(* Logix 5000 project; controller BTS01 vendor 1 type 14 code 217 rev 32.14; software revision 32.04; part 13 of 15 *)
(* tags used below, declared in another part *)
   AirBlow_Timer : TIMER;
   AirblowPB : BOOL;
   C02S01 : REAL[8];   // 5069-IF8
   C02S02 : REAL[8];   // 5069-OF8
   C02S03 : INT;   // 5069-IB16
   C02S04 : INT;   // 5069-OB16
   C02S05 : INT;   // 5069-OB16
   C02S06 : INT;   // 5069-IB16
   CIP_1_ACTIVE_CIRCUIT : DINT;
   CIP_1_RUN_LATCH : BOOL;
   CIP_1_STEP_ADV_MESSAGE : BOOL;
   CIP_RinseStep_PULSE_ENABLE : BOOL;
   CIP_WashStep_PULSE_ENABLE : BOOL;
   HMI_Alarms_Active : BOOL;
   LT1101 : DTE_SCP_W_LIM;   // Tank 1100 Level Transmitter
   LT1201 : DTE_SCP_W_LIM;   // Tank 1200 Level Transmitter
   TIMERS : TIMER[30];
   TK1100_LVL_SCP : DTE_SCP_W_LIM;   // Tank 1100 Level Remote Display
   TK1200_LVL_SCP : DTE_SCP_W_LIM;   // Tank 1200 Level Remote Display
   TransferEnabled : BOOL;
   TransferSelected : DINT;
   TransferStandby : BOOL;
   UnloadEnabled : BOOL;
   UnloadSelected : DINT;
   UnloadStandby : BOOL;
   V1002 : DTE_Air_Valve_v2;   // CIP Bypass Valve
   V1002_CIP_ENABLE : BOOL;
   V1002_CIP_PULSE : BOOL;
   V1002_Desc : STRING;
   V1002_PIDName : STRING;
   V1003 : DTE_Air_Valve_v2;   // Filler Valve
   V1003_CIP_ENABLE : BOOL;
   V1003_CIP_PULSE : BOOL;
   V1003_Desc : STRING;
   V1003_PIDName : STRING;
   V1004 : DTE_Air_Valve_v2;   // Filler Valve
   V1004_CIP_ENABLE : BOOL;
   V1004_CIP_PULSE : BOOL;
   V1004_Desc : STRING;
   V1004_PIDName : STRING;
   V1005 : DTE_Air_Valve_v2;   // Filler Valve
   V1005_CIP_ENABLE : BOOL;
   V1005_CIP_PULSE : BOOL;
   V1005_Desc : STRING;
   V1005_PIDName : STRING;
   V1006 : DTE_Air_Valve_v2;   // Filler Valve
   V1006_CIP_ENABLE : BOOL;
   V1006_CIP_PULSE : BOOL;
   V1006_Desc : STRING;
   V1006_PIDName : STRING;
   V1007 : DTE_Air_Valve_v2;   // Filler Valve
   V1007_CIP_ENABLE : BOOL;
   V1007_CIP_PULSE : BOOL;
   V1007_Desc : STRING;
   V1007_PIDName : STRING;
   V1101 : DTE_Air_Valve_v2;   // Tank 1100 Fill Valve
   V1101_CIP_ENABLE : BOOL;
   V1101_CIP_PULSE : BOOL;
   V1101_Desc : STRING;
   V1101_PIDName : STRING;
   V1102 : DTE_Air_Valve_v2;   // Tank 1100 Discharge Valve
   V1102_CIP_ENABLE : BOOL;
   V1102_CIP_PULSE : BOOL;
   V1102_Desc : STRING;
   V1102_PIDName : STRING;
   V1103 : DTE_Air_Valve_v2;   // Tank 1100 Line Valve
   V1103_CIP_ENABLE : BOOL;
   V1103_CIP_PULSE : BOOL;
   V1103_Desc : STRING;
   V1103_PIDName : STRING;
   V1201 : DTE_Air_Valve_v2;   // Tank 1200 Fill Valve
   V1201_CIP_ENABLE : BOOL;
   V1201_CIP_PULSE : BOOL;
   V1201_Desc : STRING;
   V1201_PIDName : STRING;
   V1202 : DTE_Air_Valve_v2;   // Tank 1200 Discharge Valve
   V1202_CIP_ENABLE : BOOL;
   V1202_CIP_PULSE : BOOL;
   V1202_Desc : STRING;
   V1202_PIDName : STRING;
   V1203 : DTE_Air_Valve_v2;   // Tank 1200 Line Valve
   V1203_CIP_ENABLE : BOOL;
   V1203_CIP_PULSE : BOOL;
   V1203_Desc : STRING;
   V1203_PIDName : STRING;
   VFD1001_SCP : DTE_SCP_W_LIM;   // Bowl Chopper Disc Speed Reference
   VFD1002_SCP : DTE_SCP_W_LIM;   // Dressing Tank Disc Speed Reference
   VFD1003_SCP : DTE_SCP_W_LIM;   // CIP Return Pump Speed Reference
   VFD1004_SCP : DTE_SCP_W_LIM;   // Filler CIP Return Pump Speed Reference
   VFD1101_SCP : DTE_SCP_W_LIM;   // Tank 1100 Agitator Speed Reference
   VFD1201_SCP : DTE_SCP_W_LIM;   // Tank 1200 Agitator Speed Reference
(* MainProgram, continued *)

ROUTINE R01_Digital_Input   (* ladder *)
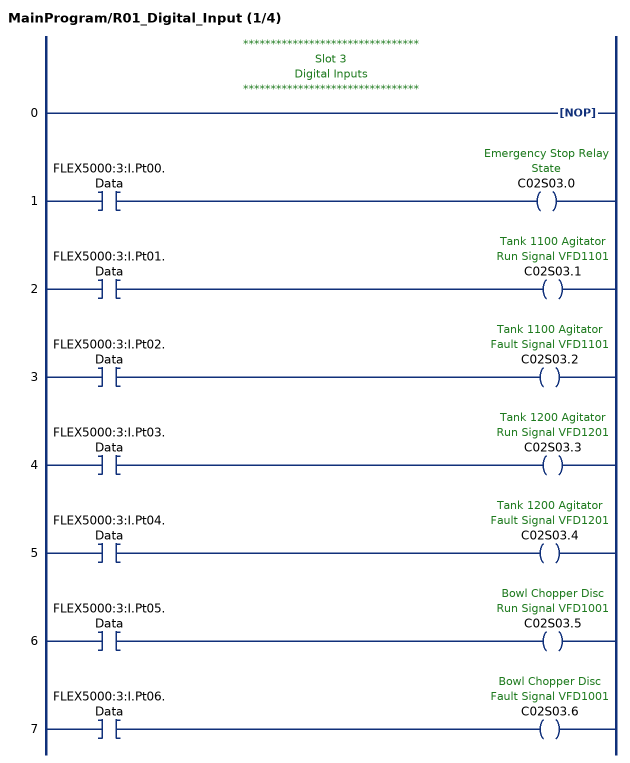
   // ********************************
   // Slot 3
   // Digital Inputs
   // ********************************
   0: NOP();
   1: XIC(FLEX5000:3:I.Pt00.Data)OTE(C02S03.0);
   2: XIC(FLEX5000:3:I.Pt01.Data)OTE(C02S03.1);
   3: XIC(FLEX5000:3:I.Pt02.Data)OTE(C02S03.2);
   4: XIC(FLEX5000:3:I.Pt03.Data)OTE(C02S03.3);
   5: XIC(FLEX5000:3:I.Pt04.Data)OTE(C02S03.4);
   6: XIC(FLEX5000:3:I.Pt05.Data)OTE(C02S03.5);
   7: XIC(FLEX5000:3:I.Pt06.Data)OTE(C02S03.6);
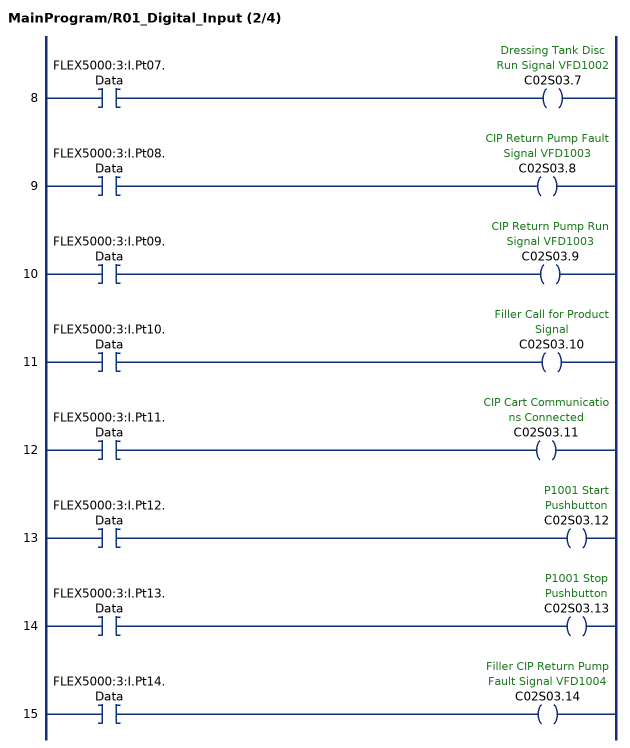
   8: XIC(FLEX5000:3:I.Pt07.Data)OTE(C02S03.7);
   9: XIC(FLEX5000:3:I.Pt08.Data)OTE(C02S03.8);
   10: XIC(FLEX5000:3:I.Pt09.Data)OTE(C02S03.9);
   11: XIC(FLEX5000:3:I.Pt10.Data)OTE(C02S03.10);
   12: XIC(FLEX5000:3:I.Pt11.Data)OTE(C02S03.11);
   13: XIC(FLEX5000:3:I.Pt12.Data)OTE(C02S03.12);
   14: XIC(FLEX5000:3:I.Pt13.Data)OTE(C02S03.13);
   15: XIC(FLEX5000:3:I.Pt14.Data)OTE(C02S03.14);
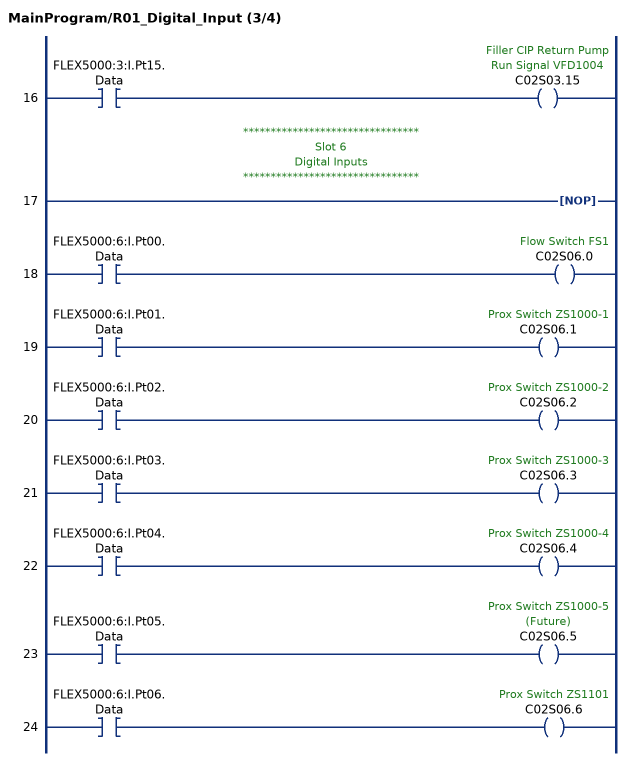
   16: XIC(FLEX5000:3:I.Pt15.Data)OTE(C02S03.15);
   // ********************************
   // Slot 6
   // Digital Inputs
   // ********************************
   17: NOP();
   18: XIC(FLEX5000:6:I.Pt00.Data)OTE(C02S06.0);
   19: XIC(FLEX5000:6:I.Pt01.Data)OTE(C02S06.1);
   20: XIC(FLEX5000:6:I.Pt02.Data)OTE(C02S06.2);
   21: XIC(FLEX5000:6:I.Pt03.Data)OTE(C02S06.3);
   22: XIC(FLEX5000:6:I.Pt04.Data)OTE(C02S06.4);
   23: XIC(FLEX5000:6:I.Pt05.Data)OTE(C02S06.5);
   24: XIC(FLEX5000:6:I.Pt06.Data)OTE(C02S06.6);
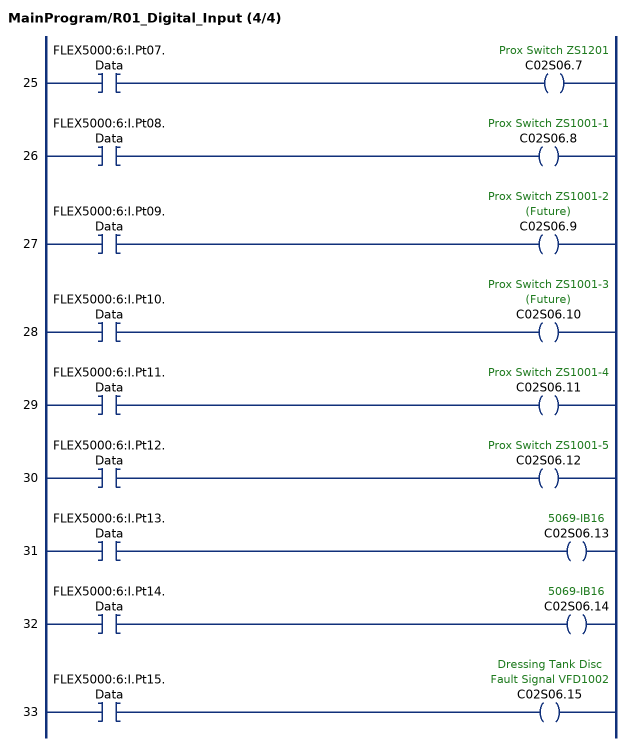
   25: XIC(FLEX5000:6:I.Pt07.Data)OTE(C02S06.7);
   26: XIC(FLEX5000:6:I.Pt08.Data)OTE(C02S06.8);
   27: XIC(FLEX5000:6:I.Pt09.Data)OTE(C02S06.9);
   28: XIC(FLEX5000:6:I.Pt10.Data)OTE(C02S06.10);
   29: XIC(FLEX5000:6:I.Pt11.Data)OTE(C02S06.11);
   30: XIC(FLEX5000:6:I.Pt12.Data)OTE(C02S06.12);
   31: XIC(FLEX5000:6:I.Pt13.Data)OTE(C02S06.13);
   32: XIC(FLEX5000:6:I.Pt14.Data)OTE(C02S06.14);
   33: XIC(FLEX5000:6:I.Pt15.Data)OTE(C02S06.15);
END_ROUTINE

ROUTINE R02_Digital_Output   (* ladder *)
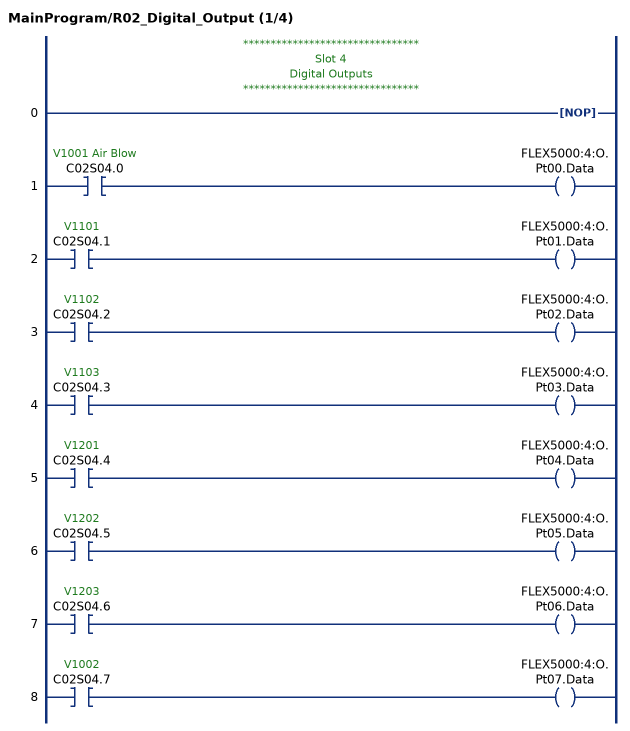
   // ********************************
   // Slot 4
   // Digital Outputs
   // ********************************
   0: NOP();
   1: XIC(C02S04.0)OTE(FLEX5000:4:O.Pt00.Data);
   2: XIC(C02S04.1)OTE(FLEX5000:4:O.Pt01.Data);
   3: XIC(C02S04.2)OTE(FLEX5000:4:O.Pt02.Data);
   4: XIC(C02S04.3)OTE(FLEX5000:4:O.Pt03.Data);
   5: XIC(C02S04.4)OTE(FLEX5000:4:O.Pt04.Data);
   6: XIC(C02S04.5)OTE(FLEX5000:4:O.Pt05.Data);
   7: XIC(C02S04.6)OTE(FLEX5000:4:O.Pt06.Data);
   8: XIC(C02S04.7)OTE(FLEX5000:4:O.Pt07.Data);
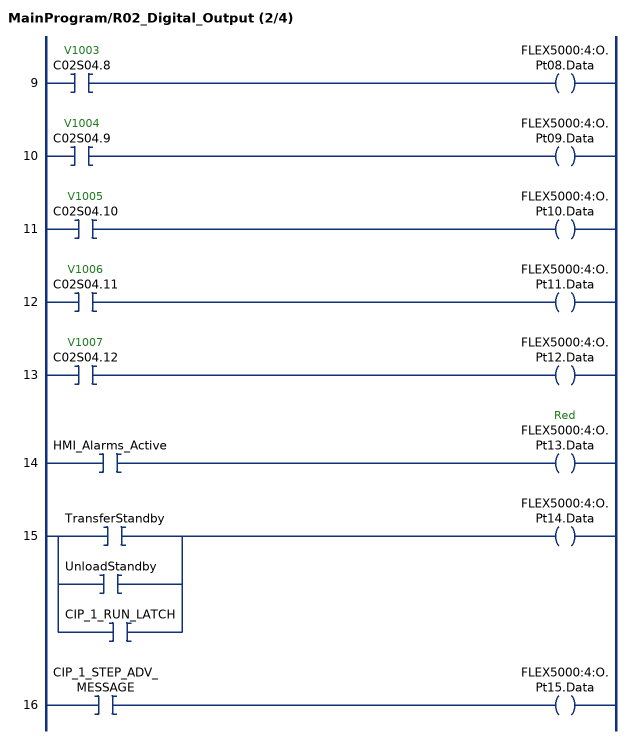
   9: XIC(C02S04.8)OTE(FLEX5000:4:O.Pt08.Data);
   10: XIC(C02S04.9)OTE(FLEX5000:4:O.Pt09.Data);
   11: XIC(C02S04.10)OTE(FLEX5000:4:O.Pt10.Data);
   12: XIC(C02S04.11)OTE(FLEX5000:4:O.Pt11.Data);
   13: XIC(C02S04.12)OTE(FLEX5000:4:O.Pt12.Data);
   14: XIC(HMI_Alarms_Active)OTE(FLEX5000:4:O.Pt13.Data);
   15: [XIC(TransferStandby) ,XIC(UnloadStandby) ,XIC(CIP_1_RUN_LATCH) ]OTE(FLEX5000:4:O.Pt14.Data);
   16: XIC(CIP_1_STEP_ADV_MESSAGE)OTE(FLEX5000:4:O.Pt15.Data);
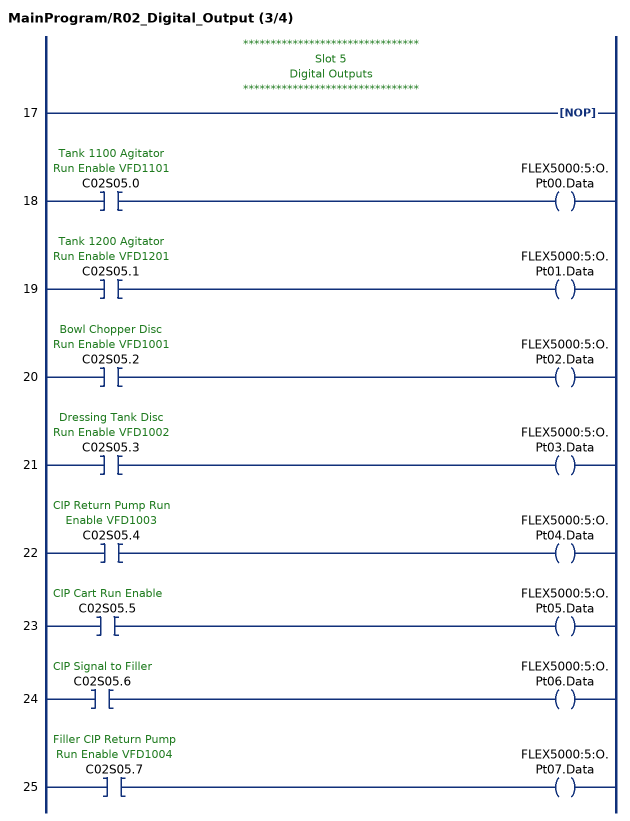
   // ********************************
   // Slot 5
   // Digital Outputs
   // ********************************
   17: NOP();
   18: XIC(C02S05.0)OTE(FLEX5000:5:O.Pt00.Data);
   19: XIC(C02S05.1)OTE(FLEX5000:5:O.Pt01.Data);
   20: XIC(C02S05.2)OTE(FLEX5000:5:O.Pt02.Data);
   21: XIC(C02S05.3)OTE(FLEX5000:5:O.Pt03.Data);
   22: XIC(C02S05.4)OTE(FLEX5000:5:O.Pt04.Data);
   23: XIC(C02S05.5)OTE(FLEX5000:5:O.Pt05.Data);
   24: XIC(C02S05.6)OTE(FLEX5000:5:O.Pt06.Data);
   25: XIC(C02S05.7)OTE(FLEX5000:5:O.Pt07.Data);
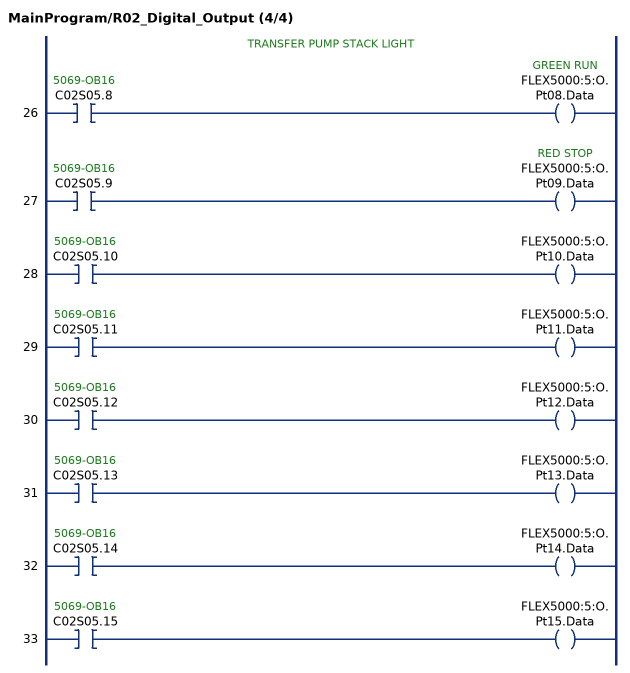
   // TRANSFER PUMP STACK LIGHT
   26: XIC(C02S05.8)OTE(FLEX5000:5:O.Pt08.Data);
   27: XIC(C02S05.9)OTE(FLEX5000:5:O.Pt09.Data);
   28: XIC(C02S05.10)OTE(FLEX5000:5:O.Pt10.Data);
   29: XIC(C02S05.11)OTE(FLEX5000:5:O.Pt11.Data);
   30: XIC(C02S05.12)OTE(FLEX5000:5:O.Pt12.Data);
   31: XIC(C02S05.13)OTE(FLEX5000:5:O.Pt13.Data);
   32: XIC(C02S05.14)OTE(FLEX5000:5:O.Pt14.Data);
   33: XIC(C02S05.15)OTE(FLEX5000:5:O.Pt15.Data);
END_ROUTINE

ROUTINE R03_Analog_Input   (* ladder *)
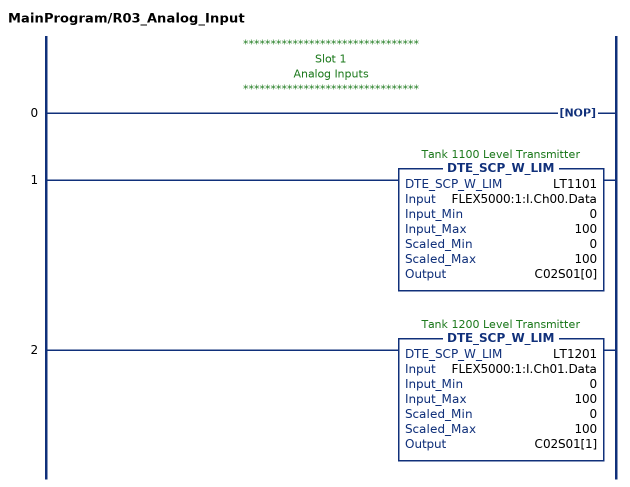
   // ********************************
   // Slot 1
   // Analog Inputs
   // ********************************
   0: NOP();
   1: DTE_SCP_W_LIM(LT1101,FLEX5000:1:I.Ch00.Data,0,100,0,100,C02S01[0]);
   2: DTE_SCP_W_LIM(LT1201,FLEX5000:1:I.Ch01.Data,0,100,0,100,C02S01[1]);
END_ROUTINE

ROUTINE R04_Analog_Output   (* ladder *)
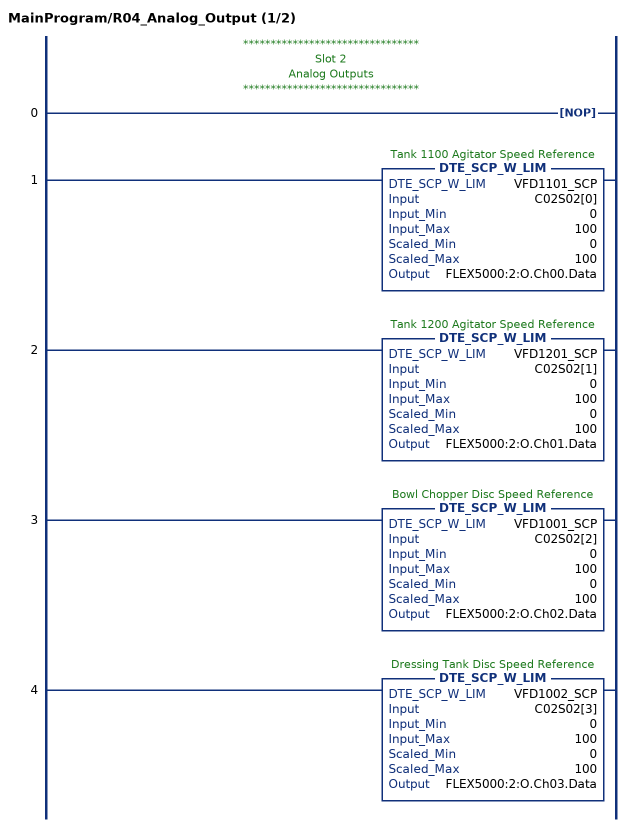
   // ********************************
   // Slot 2
   // Analog Outputs
   // ********************************
   0: NOP();
   1: DTE_SCP_W_LIM(VFD1101_SCP,C02S02[0],0,100,0,100,FLEX5000:2:O.Ch00.Data);
   2: DTE_SCP_W_LIM(VFD1201_SCP,C02S02[1],0,100,0,100,FLEX5000:2:O.Ch01.Data);
   3: DTE_SCP_W_LIM(VFD1001_SCP,C02S02[2],0,100,0,100,FLEX5000:2:O.Ch02.Data);
   4: DTE_SCP_W_LIM(VFD1002_SCP,C02S02[3],0,100,0,100,FLEX5000:2:O.Ch03.Data);
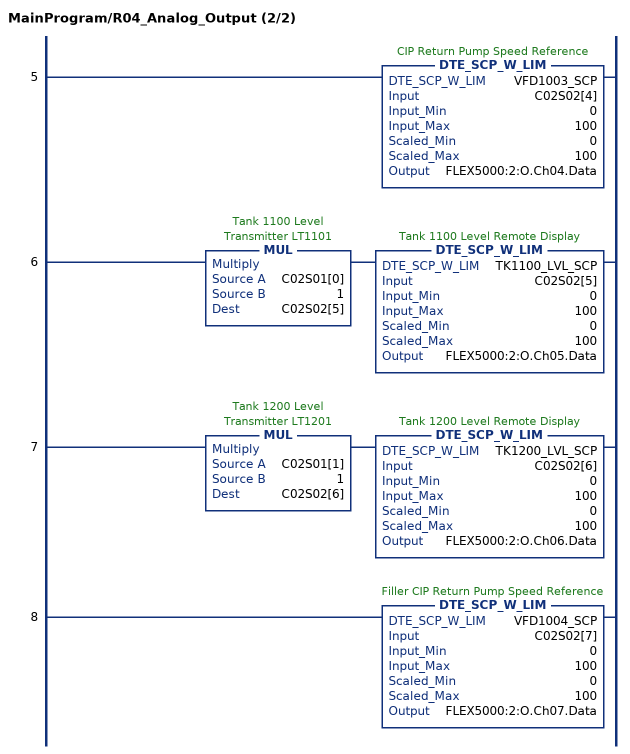
   5: DTE_SCP_W_LIM(VFD1003_SCP,C02S02[4],0,100,0,100,FLEX5000:2:O.Ch04.Data);
   6: MUL(C02S01[0],1,C02S02[5])DTE_SCP_W_LIM(TK1100_LVL_SCP,C02S02[5],0,100,0,100,FLEX5000:2:O.Ch05.Data);
   7: MUL(C02S01[1],1,C02S02[6])DTE_SCP_W_LIM(TK1200_LVL_SCP,C02S02[6],0,100,0,100,FLEX5000:2:O.Ch06.Data);
   8: DTE_SCP_W_LIM(VFD1004_SCP,C02S02[7],0,100,0,100,FLEX5000:2:O.Ch07.Data);
END_ROUTINE

ROUTINE R05_Valves   (* ladder *)
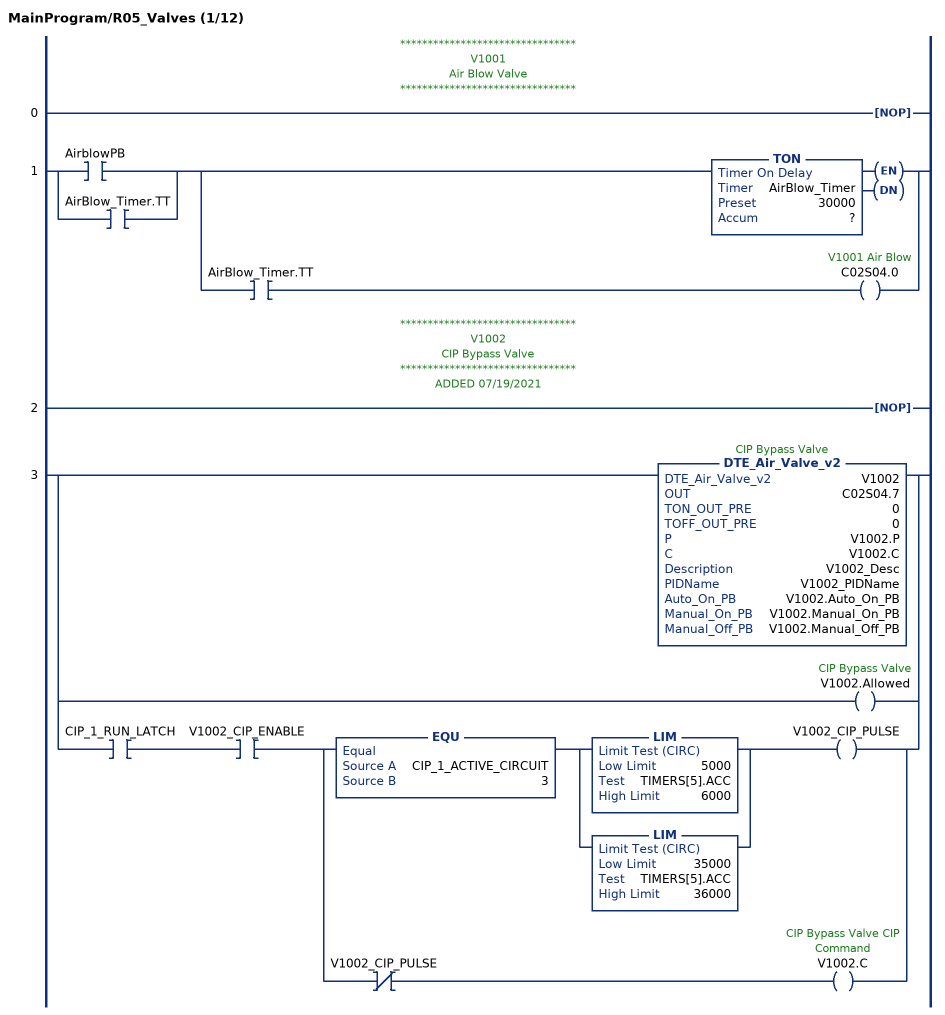
   // ********************************
   // V1001
   // Air Blow Valve
   // ********************************
   0: NOP();
   1: [XIC(AirblowPB) ,XIC(AirBlow_Timer.TT) ][TON(AirBlow_Timer,?,?) ,XIC(AirBlow_Timer.TT) OTE(C02S04.0) ];
   // ********************************
   // V1002
   // CIP Bypass Valve
   // ********************************
   // ADDED 07/19/2021
   2: NOP();
   3: [DTE_Air_Valve_v2(V1002,C02S04.7,0,0,V1002.P,V1002.C,V1002_Desc,V1002_PIDName,V1002.Auto_On_PB,V1002.Manual_On_PB,V1002.Manual_Off_PB) ,OTE(V1002.Allowed) ,XIC(CIP_1_RUN_LATCH) XIC(V1002_CIP_ENABLE) [EQU(CIP_1_ACTIVE_CIRCUIT,3) [LIM(5000,TIMERS[5].ACC,6000) ,LIM(35000,TIMERS[5].ACC,36000) ] OTE(V1002_CIP_PULSE) ,XIO(V1002_CIP_PULSE) OTE(V1002.C) ] ];
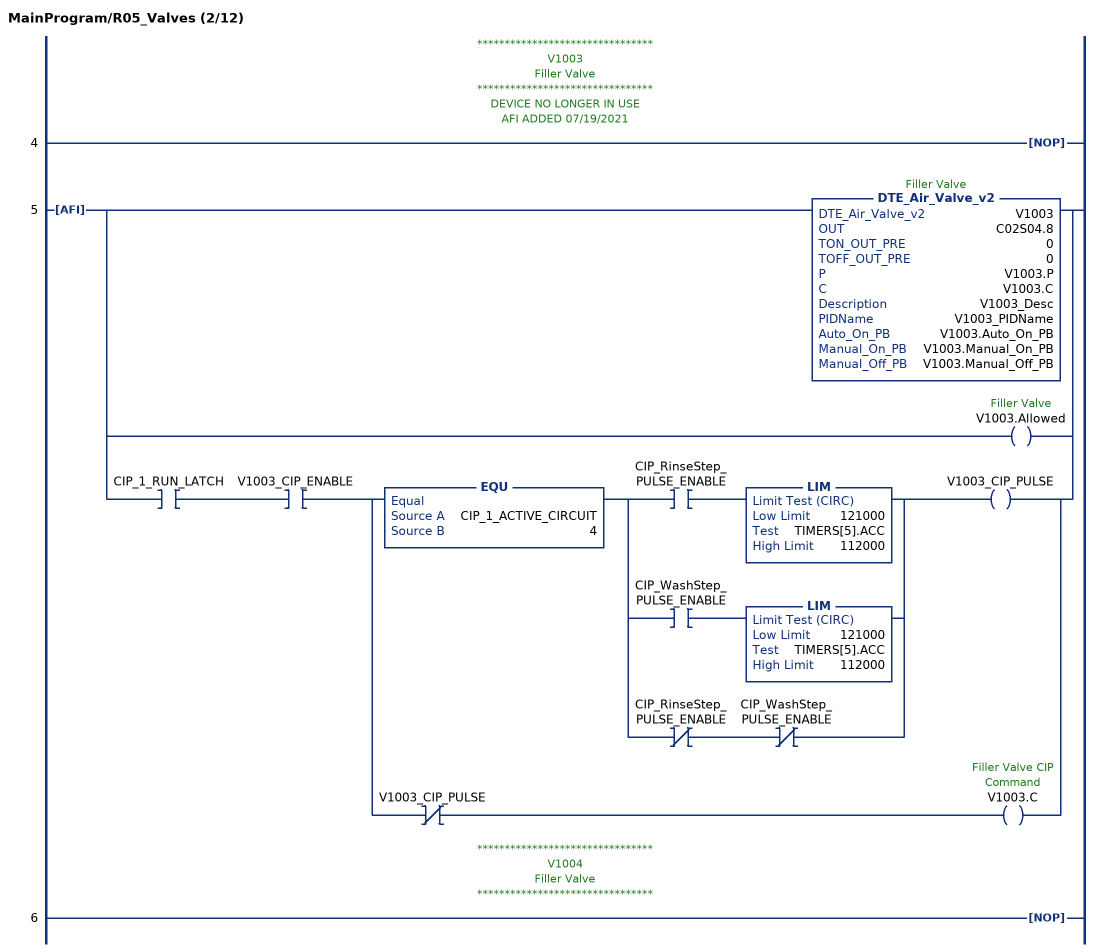
   // ********************************
   // V1003
   // Filler Valve
   // ********************************
   // DEVICE NO LONGER IN USE
   // AFI ADDED 07/19/2021
   4: NOP();
   5: AFI()[DTE_Air_Valve_v2(V1003,C02S04.8,0,0,V1003.P,V1003.C,V1003_Desc,V1003_PIDName,V1003.Auto_On_PB,V1003.Manual_On_PB,V1003.Manual_Off_PB) ,OTE(V1003.Allowed) ,XIC(CIP_1_RUN_LATCH) XIC(V1003_CIP_ENABLE) [EQU(CIP_1_ACTIVE_CIRCUIT,4) [XIC(CIP_RinseStep_PULSE_ENABLE) LIM(121000,TIMERS[5].ACC,112000) ,XIC(CIP_WashStep_PULSE_ENABLE) LIM(121000,TIMERS[5].ACC,112000) ,XIO(CIP_RinseStep_PULSE_ENABLE) XIO(CIP_WashStep_PULSE_ENABLE) ] OTE(V1003_CIP_PULSE) ,XIO(V1003_CIP_PULSE) OTE(V1003.C) ] ];
   // ********************************
   // V1004
   // Filler Valve
   // ********************************
   6: NOP();
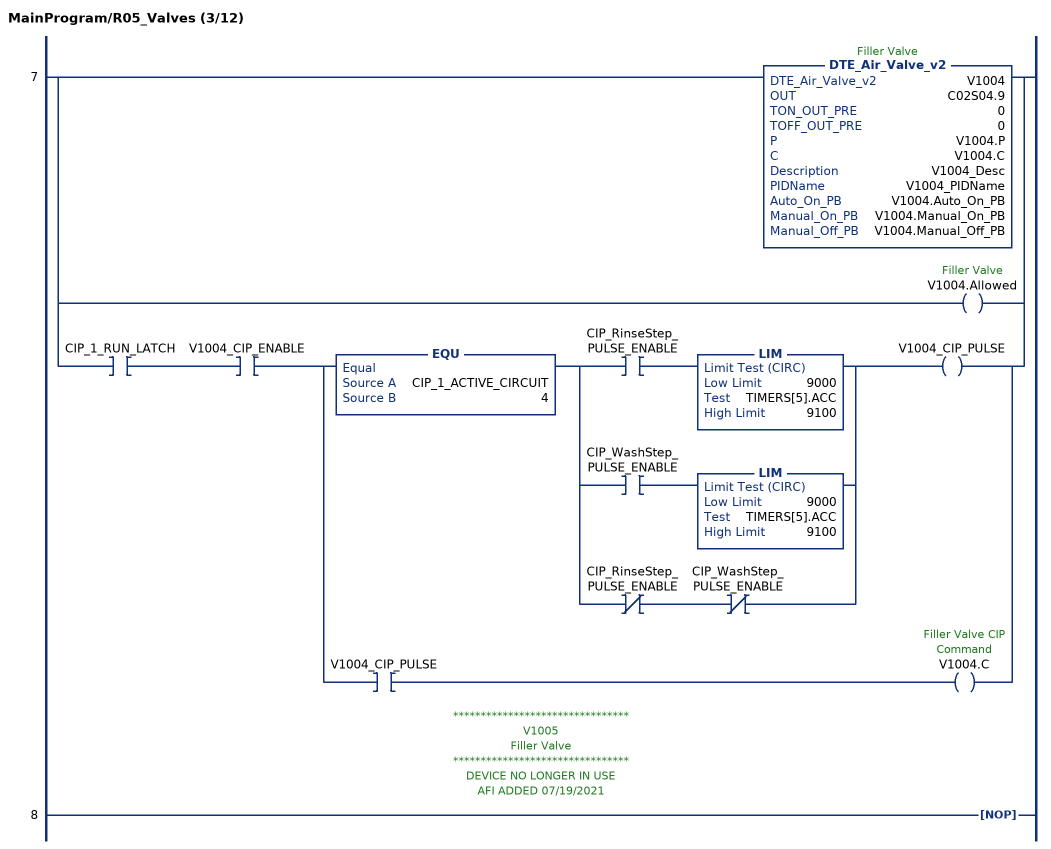
   7: [DTE_Air_Valve_v2(V1004,C02S04.9,0,0,V1004.P,V1004.C,V1004_Desc,V1004_PIDName,V1004.Auto_On_PB,V1004.Manual_On_PB,V1004.Manual_Off_PB) ,OTE(V1004.Allowed) ,XIC(CIP_1_RUN_LATCH) XIC(V1004_CIP_ENABLE) [EQU(CIP_1_ACTIVE_CIRCUIT,4) [XIC(CIP_RinseStep_PULSE_ENABLE) LIM(9000,TIMERS[5].ACC,9100) ,XIC(CIP_WashStep_PULSE_ENABLE) LIM(9000,TIMERS[5].ACC,9100) ,XIO(CIP_RinseStep_PULSE_ENABLE) XIO(CIP_WashStep_PULSE_ENABLE) ] OTE(V1004_CIP_PULSE) ,XIC(V1004_CIP_PULSE) OTE(V1004.C) ] ];
   // ********************************
   // V1005
   // Filler Valve
   // ********************************
   // DEVICE NO LONGER IN USE
   // AFI ADDED 07/19/2021
   8: NOP();
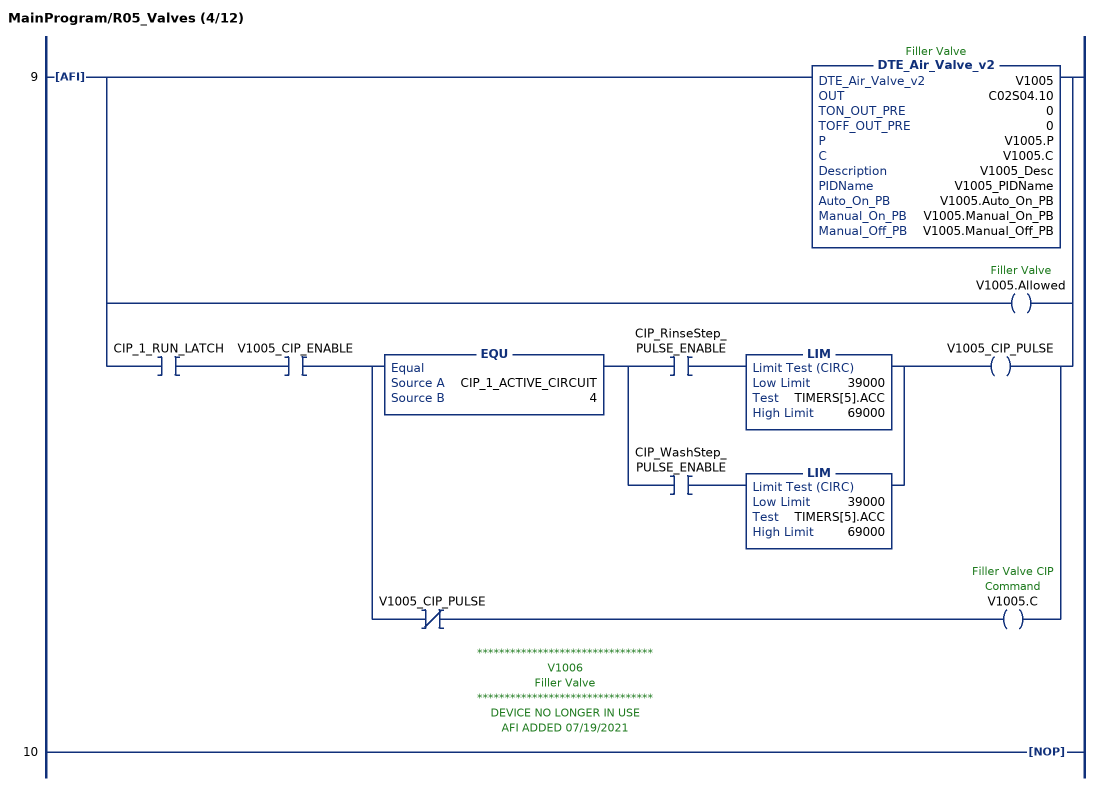
   9: AFI()[DTE_Air_Valve_v2(V1005,C02S04.10,0,0,V1005.P,V1005.C,V1005_Desc,V1005_PIDName,V1005.Auto_On_PB,V1005.Manual_On_PB,V1005.Manual_Off_PB) ,OTE(V1005.Allowed) ,XIC(CIP_1_RUN_LATCH) XIC(V1005_CIP_ENABLE) [EQU(CIP_1_ACTIVE_CIRCUIT,4) [XIC(CIP_RinseStep_PULSE_ENABLE) LIM(39000,TIMERS[5].ACC,69000) ,XIC(CIP_WashStep_PULSE_ENABLE) LIM(39000,TIMERS[5].ACC,69000) ] OTE(V1005_CIP_PULSE) ,XIO(V1005_CIP_PULSE) OTE(V1005.C) ] ];
   // ********************************
   // V1006
   // Filler Valve
   // ********************************
   // DEVICE NO LONGER IN USE
   // AFI ADDED 07/19/2021
   10: NOP();
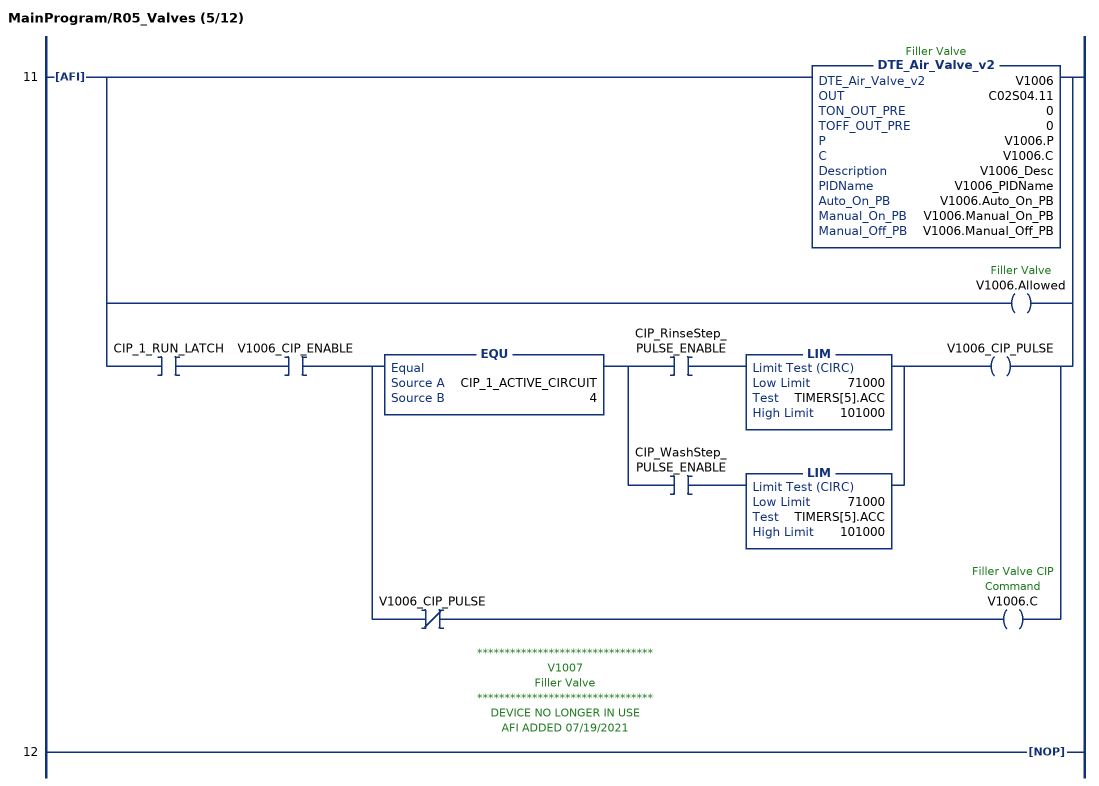
   11: AFI()[DTE_Air_Valve_v2(V1006,C02S04.11,0,0,V1006.P,V1006.C,V1006_Desc,V1006_PIDName,V1006.Auto_On_PB,V1006.Manual_On_PB,V1006.Manual_Off_PB) ,OTE(V1006.Allowed) ,XIC(CIP_1_RUN_LATCH) XIC(V1006_CIP_ENABLE) [EQU(CIP_1_ACTIVE_CIRCUIT,4) [XIC(CIP_RinseStep_PULSE_ENABLE) LIM(71000,TIMERS[5].ACC,101000) ,XIC(CIP_WashStep_PULSE_ENABLE) LIM(71000,TIMERS[5].ACC,101000) ] OTE(V1006_CIP_PULSE) ,XIO(V1006_CIP_PULSE) OTE(V1006.C) ] ];
   // ********************************
   // V1007
   // Filler Valve
   // ********************************
   // DEVICE NO LONGER IN USE
   // AFI ADDED 07/19/2021
   12: NOP();
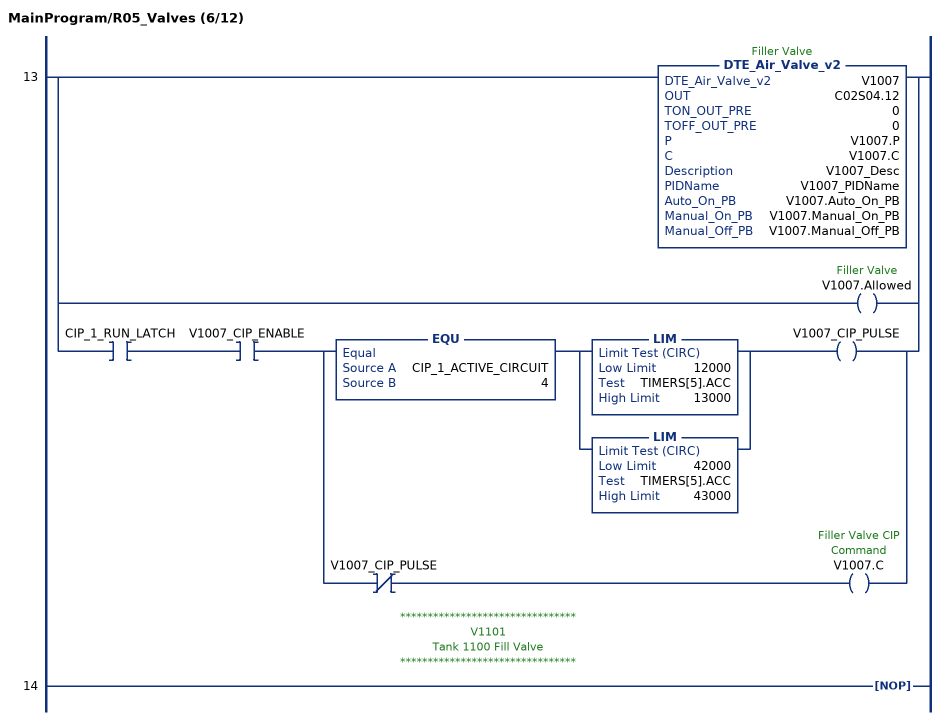
   13: [DTE_Air_Valve_v2(V1007,C02S04.12,0,0,V1007.P,V1007.C,V1007_Desc,V1007_PIDName,V1007.Auto_On_PB,V1007.Manual_On_PB,V1007.Manual_Off_PB) ,OTE(V1007.Allowed) ,XIC(CIP_1_RUN_LATCH) XIC(V1007_CIP_ENABLE) [EQU(CIP_1_ACTIVE_CIRCUIT,4) [LIM(12000,TIMERS[5].ACC,13000) ,LIM(42000,TIMERS[5].ACC,43000) ] OTE(V1007_CIP_PULSE) ,XIO(V1007_CIP_PULSE) OTE(V1007.C) ] ];
   // ********************************
   // V1101
   // Tank 1100 Fill Valve
   // ********************************
   14: NOP();
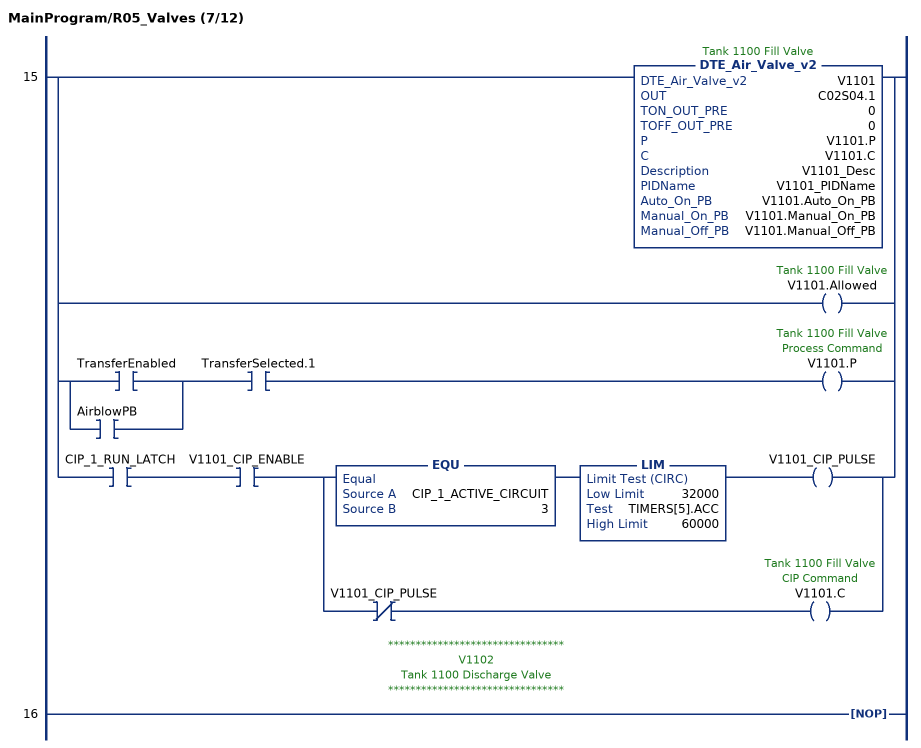
   15: [DTE_Air_Valve_v2(V1101,C02S04.1,0,0,V1101.P,V1101.C,V1101_Desc,V1101_PIDName,V1101.Auto_On_PB,V1101.Manual_On_PB,V1101.Manual_Off_PB) ,OTE(V1101.Allowed) ,[XIC(TransferEnabled) ,XIC(AirblowPB) ] XIC(TransferSelected.1) OTE(V1101.P) ,XIC(CIP_1_RUN_LATCH) XIC(V1101_CIP_ENABLE) [EQU(CIP_1_ACTIVE_CIRCUIT,3) LIM(32000,TIMERS[5].ACC,60000) OTE(V1101_CIP_PULSE) ,XIO(V1101_CIP_PULSE) OTE(V1101.C) ] ];
   // ********************************
   // V1102
   // Tank 1100 Discharge Valve
   // ********************************
   16: NOP();
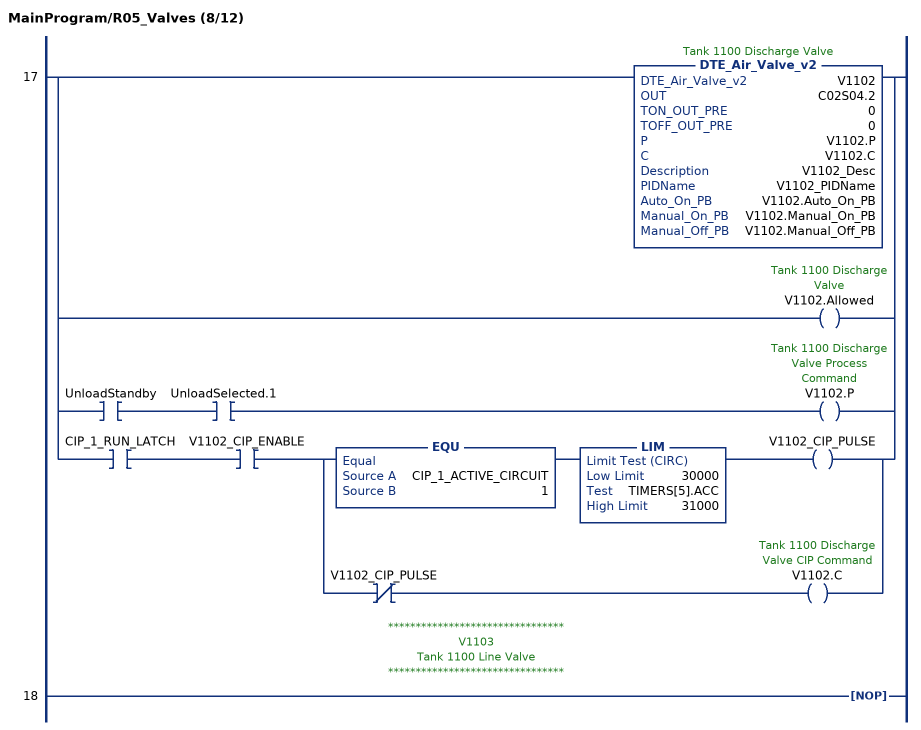
   17: [DTE_Air_Valve_v2(V1102,C02S04.2,0,0,V1102.P,V1102.C,V1102_Desc,V1102_PIDName,V1102.Auto_On_PB,V1102.Manual_On_PB,V1102.Manual_Off_PB) ,OTE(V1102.Allowed) ,XIC(UnloadStandby) XIC(UnloadSelected.1) OTE(V1102.P) ,XIC(CIP_1_RUN_LATCH) XIC(V1102_CIP_ENABLE) [EQU(CIP_1_ACTIVE_CIRCUIT,1) LIM(30000,TIMERS[5].ACC,31000) OTE(V1102_CIP_PULSE) ,XIO(V1102_CIP_PULSE) OTE(V1102.C) ] ];
   // ********************************
   // V1103
   // Tank 1100 Line Valve
   // ********************************
   18: NOP();
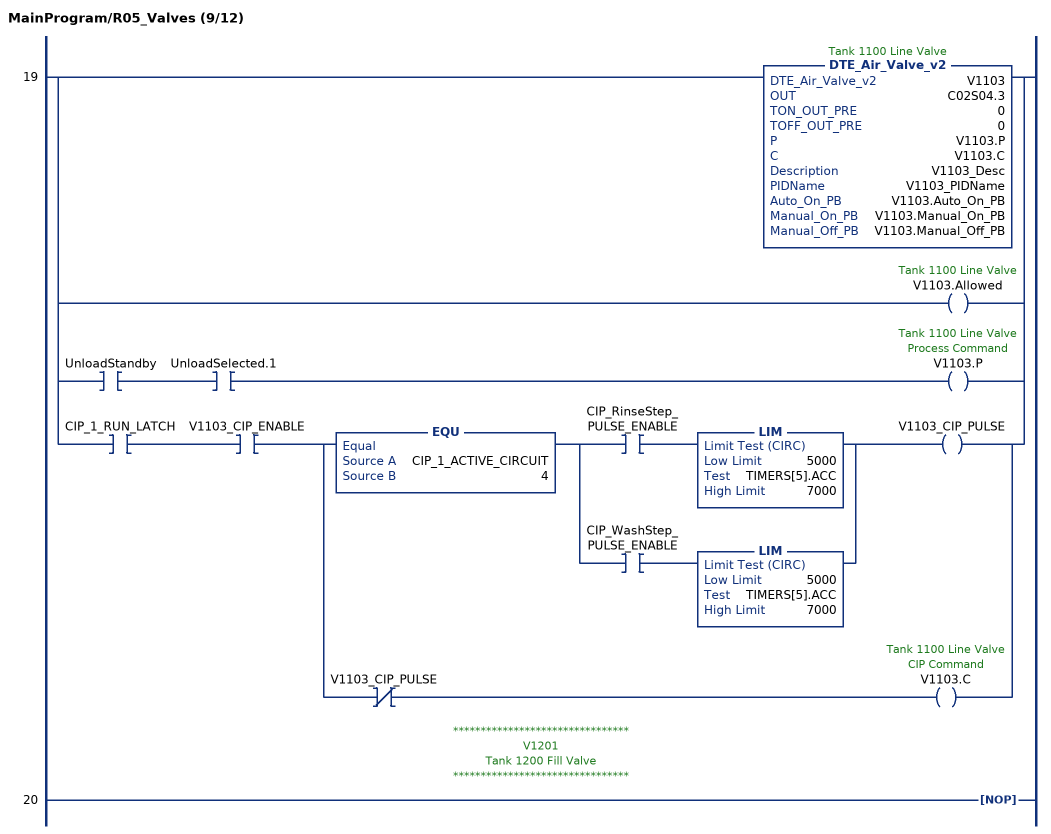
   19: [DTE_Air_Valve_v2(V1103,C02S04.3,0,0,V1103.P,V1103.C,V1103_Desc,V1103_PIDName,V1103.Auto_On_PB,V1103.Manual_On_PB,V1103.Manual_Off_PB) ,OTE(V1103.Allowed) ,XIC(UnloadStandby) XIC(UnloadSelected.1) OTE(V1103.P) ,XIC(CIP_1_RUN_LATCH) XIC(V1103_CIP_ENABLE) [EQU(CIP_1_ACTIVE_CIRCUIT,4) [XIC(CIP_RinseStep_PULSE_ENABLE) LIM(5000,TIMERS[5].ACC,7000) ,XIC(CIP_WashStep_PULSE_ENABLE) LIM(5000,TIMERS[5].ACC,7000) ] OTE(V1103_CIP_PULSE) ,XIO(V1103_CIP_PULSE) OTE(V1103.C) ] ];
   // ********************************
   // V1201
   // Tank 1200 Fill Valve
   // ********************************
   20: NOP();
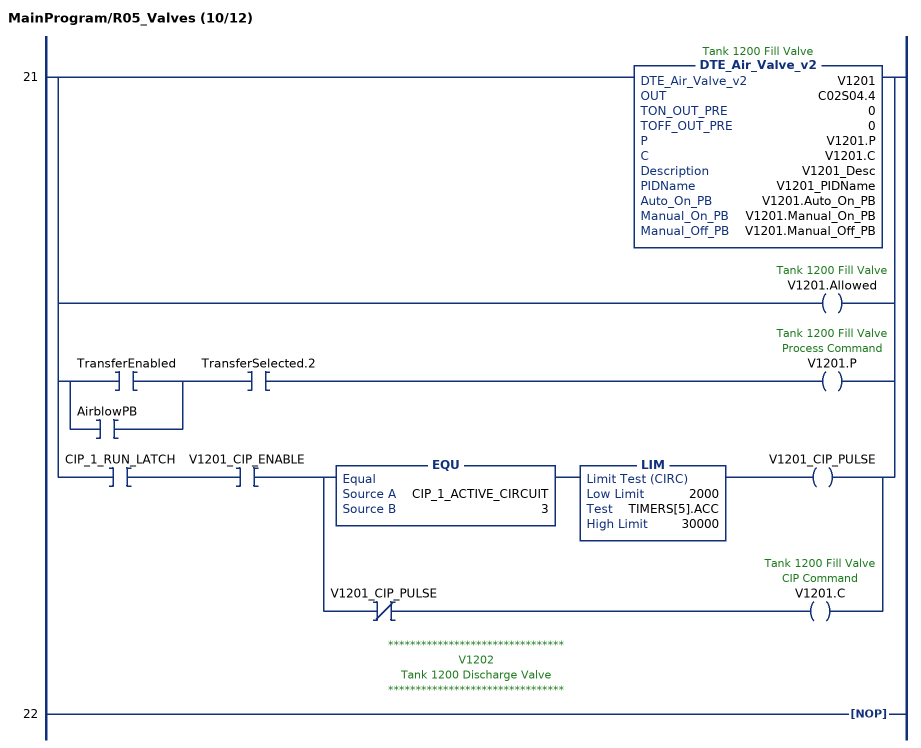
   21: [DTE_Air_Valve_v2(V1201,C02S04.4,0,0,V1201.P,V1201.C,V1201_Desc,V1201_PIDName,V1201.Auto_On_PB,V1201.Manual_On_PB,V1201.Manual_Off_PB) ,OTE(V1201.Allowed) ,[XIC(TransferEnabled) ,XIC(AirblowPB) ] XIC(TransferSelected.2) OTE(V1201.P) ,XIC(CIP_1_RUN_LATCH) XIC(V1201_CIP_ENABLE) [EQU(CIP_1_ACTIVE_CIRCUIT,3) LIM(2000,TIMERS[5].ACC,30000) OTE(V1201_CIP_PULSE) ,XIO(V1201_CIP_PULSE) OTE(V1201.C) ] ];
   // ********************************
   // V1202
   // Tank 1200 Discharge Valve
   // ********************************
   22: NOP();
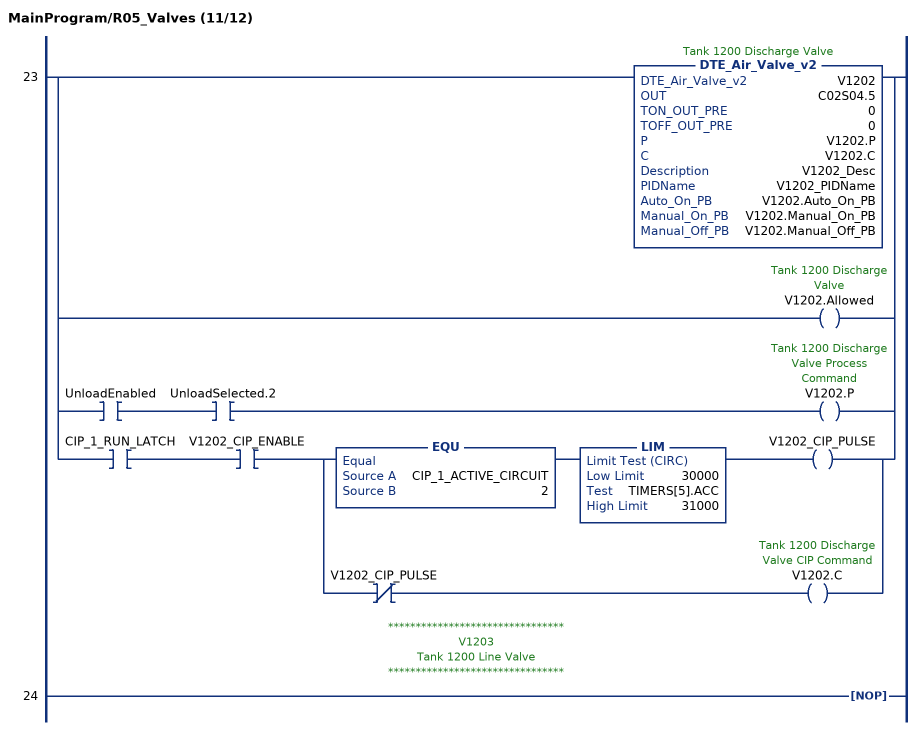
   23: [DTE_Air_Valve_v2(V1202,C02S04.5,0,0,V1202.P,V1202.C,V1202_Desc,V1202_PIDName,V1202.Auto_On_PB,V1202.Manual_On_PB,V1202.Manual_Off_PB) ,OTE(V1202.Allowed) ,XIC(UnloadEnabled) XIC(UnloadSelected.2) OTE(V1202.P) ,XIC(CIP_1_RUN_LATCH) XIC(V1202_CIP_ENABLE) [EQU(CIP_1_ACTIVE_CIRCUIT,2) LIM(30000,TIMERS[5].ACC,31000) OTE(V1202_CIP_PULSE) ,XIO(V1202_CIP_PULSE) OTE(V1202.C) ] ];
   // ********************************
   // V1203
   // Tank 1200 Line Valve
   // ********************************
   24: NOP();
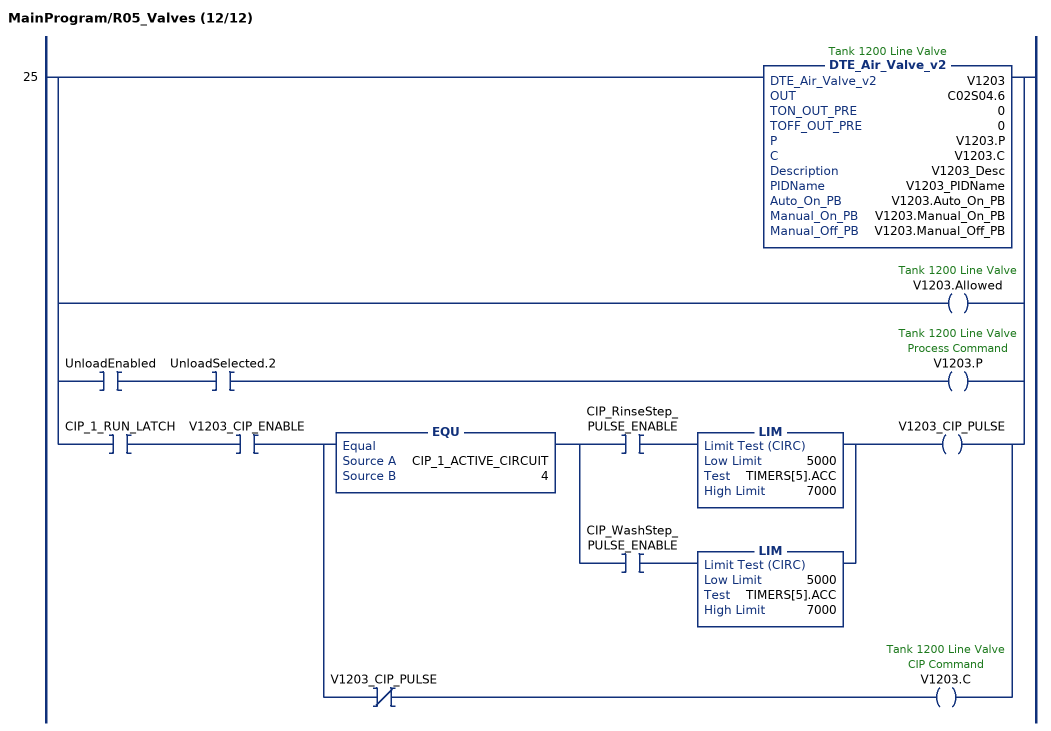
   25: [DTE_Air_Valve_v2(V1203,C02S04.6,0,0,V1203.P,V1203.C,V1203_Desc,V1203_PIDName,V1203.Auto_On_PB,V1203.Manual_On_PB,V1203.Manual_Off_PB) ,OTE(V1203.Allowed) ,XIC(UnloadEnabled) XIC(UnloadSelected.2) OTE(V1203.P) ,XIC(CIP_1_RUN_LATCH) XIC(V1203_CIP_ENABLE) [EQU(CIP_1_ACTIVE_CIRCUIT,4) [XIC(CIP_RinseStep_PULSE_ENABLE) LIM(5000,TIMERS[5].ACC,7000) ,XIC(CIP_WashStep_PULSE_ENABLE) LIM(5000,TIMERS[5].ACC,7000) ] OTE(V1203_CIP_PULSE) ,XIO(V1203_CIP_PULSE) OTE(V1203.C) ] ];
END_ROUTINE
